INTERFACE ITF_ControlE_TE2_HMI_Connector EXTENDS ITF_BaseControlElement_HMI_Connector

END_INTERFACE

(* stored: Version 1.1.0.1, ProductVersion 3.1.4024.15
   Itf ITF_ControlE_TE2_HMI_Connector: Id {36eb920a-5278-42ed-a7c4-9f2b3c3df23f} *)
